Staubli VAL3: BINTODEC.pgx

public program binToDec(string x_value, num& x_return[])
// change binary string to num variable (e.g. "1001" => 9)
  local num l_bit
begin
  x_return=0
  for l_bit=(len(x_value)-1) to 0 step -1
    if mid(x_value,1,l_bit)=="1"
      x_return=x_return+exp(((len(x_value)-1)-l_bit)*ln(2))
    endIf
  endFor
  if bDebug
    putln("binToDec(): "+x_value+" => "+toString("0.0",x_return))
  endIf
end
